(* IEC 61131-3 sources: Lasal/CPU_5344_V01/Class/baseToolSettingsMpsControl, 1 file *)

(* ---- baseToolSettingsMpsControl.st ---- *)
(*!
<Class
	Name               = "baseToolSettingsMpsControl"
	Revision           = "1.0"
	RealtimeTask       = "false"
	CyclicTask         = "false"
	BackgroundTask     = "false"
	Sigmatek           = "false"
	OSInterface        = "false"
	HighPriority       = "false"
	Automatic          = "false"
	UpdateMode         = "Prescan"
	SharedCommandTable = "true"
	Objectsize         = "(284,120)">
	<Channels>
		<Server Name="amountOfSettings" Visualized="true" Initialize="true" DefValue="4" WriteProtected="true" Retentive="false"/>
		<Server Name="ClassSvr" Visualized="false" Initialize="false" WriteProtected="true" Retentive="false"/>
		<Server Name="Name" Class="StringRAM" Visualized="true" Remotely="true" Initialize="true" WriteProtected="false" Retentive="false"/>
		<Server Name="plane" Visualized="true" Initialize="true" DefValue="right" WriteProtected="true" Retentive="false"/>
		<Server Name="toolType" Visualized="true" Initialize="true" DefValue="9" WriteProtected="true" Retentive="false"/>
		<Client Name="unitName" Required="true" Internal="true"/>
	</Channels>
	<Network Name="baseToolSettingsMpsControl">
		<!-- List of Components in this network -->
		<Components>
			<Object
				Name       = "unitName"
				Class      = "StringRAM"
				Position   = "(150,600)"
				Visualized = "true"
				Remotely   = "true">
				<Channels>
					<Server Name="Data"/>
					<Client Name="SingleRealloc" Value="1"/>
					<Client Name="UseFile" Value="1"/>
				</Channels>
			</Object>
		</Components>
		<Comments>
		</Comments>
		<!-- List of Connections in this network -->
		<Connections>
			<Connection Source="this.unitName" Destination="unitName.Data"/>
			<Connection Source="this.Name" Destination="unitName.Data" Vertices="(848,330),(676,690),"/>
		</Connections>
		<!-- Headerfiles -->
		<Options>
		</Options>
	</Network>
</Class>
*)
baseToolSettingsMpsControl : CLASS
  //Servers:
	ClassSvr 	: SvrChCmd_DINT;
	toolType 	: SvrCh_pcUnitTypes;
	Name 	: SvrChCmd_UDINT;
	plane 	: SvrCh_pcPlaneType;
	amountOfSettings 	: SvrCh_DINT;
  //Clients:
	unitName 	: CltChCmd_StringRAM;
  //Variables:
  //Functions:

	FUNCTION VIRTUAL GLOBAL Name::Read
		VAR_OUTPUT
			output (EAX) 	: UDINT;
		END_VAR;

	FUNCTION VIRTUAL GLOBAL Name::Write
		VAR_INPUT
			input (EAX) 	: UDINT;
		END_VAR
		VAR_OUTPUT
			result (EAX) 	: UDINT;
		END_VAR;
  //Tables:
	FUNCTION @STD
		VAR_OUTPUT
			ret_code	: CONFSTATES;
		END_VAR;
	FUNCTION GLOBAL TAB @CT_;
END_CLASS;

#pragma using StringRAM

// JdK 6-2-2020: baseToolSettingsMpsControl created for first test to read in settings to pc
// at this moment the class is only for storage off fixed machine data for all tools, is overrided for real tool

FUNCTION VIRTUAL GLOBAL baseToolSettingsMpsControl::Name::Read
	VAR_OUTPUT
		output (EAX) 	: UDINT;
	END_VAR

	Name := unitName.Data.Read();
	output := Name;

END_FUNCTION

FUNCTION VIRTUAL GLOBAL baseToolSettingsMpsControl::Name::Write
	VAR_INPUT
		input (EAX) 	: UDINT;
	END_VAR
	VAR_OUTPUT
		result (EAX) 	: UDINT;
	END_VAR

	Name := input;
	result := (unitName.Data.Write(Name))$UDINT;

END_FUNCTION
